TYPE ST_PowerControl_SocDroopParams :
STRUCT
	enable				: BOOL := TRUE;
	SocMinDroopStart	: REAL := 20; // at XX%, frequency is shifted linearly down with the actual SOC towards 0%.
	SocMaxDroopStart	: REAL := 80; // at XX%, frequency is shifted linearly up with the actual SOC towards 100%.
END_STRUCT
END_TYPE

(* stored: Version 1.1.0.1, ProductVersion 3.1.4026.18
   DUT ST_PowerControl_SocDroopParams: Id {03ed2776-4005-4b6f-abaf-f6dce5869e8f} *)
